KUKA KRL program: SET_AXIS_MAXDELTA.src

&ACCESS RVO
&REL 6
&PARAM TEMPLATE = C:\KRC\Roboter\Template\FunctionVorgabe
&PARAM EDITMASK = *
DEFFCT BOOL SET_AXIS_MAXDELTA( A1_VAL:IN, A2_VAL:IN, A3_VAL:IN, A4_VAL:IN, A5_VAL:IN, A6_VAL:IN, E1_VAL:IN)

REAL A1_VAL, A2_VAL, A3_VAL
REAL A4_VAL, A5_VAL, A6_VAL
REAL E1_VAL

$STIFFNESS.AXISMAXDELTA.A1 = A1_VAL
$STIFFNESS.AXISMAXDELTA.A2 = A2_VAL
$STIFFNESS.AXISMAXDELTA.A3 = A3_VAL
$STIFFNESS.AXISMAXDELTA.A4 = A4_VAL
$STIFFNESS.AXISMAXDELTA.A5 = A5_VAL
$STIFFNESS.AXISMAXDELTA.A6 = A6_VAL
$STIFFNESS.AXISMAXDELTA.E1 = E1_VAL

$STIFFNESS.COMMIT = TRUE

RETURN TRUE

ENDFCT
